FUNCTION_BLOCK Q_ChildPosition (* Command change child position ( Part 6 - F.16 ) *)
  (* Standard: ISO 11783-6; Description: The Change Child Location command is used to change the absolute position of an object. Return values iso_s16 - E_NO_ERR - OK - E_OVERFLOW - buffer overflow - E_NOACT - Command not possible in current state - E_NO_INSTANCE - No VT client available *)
  (* Version 1.0, 2022-07-08, franz *)
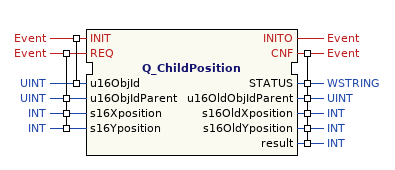
  EVENT_INPUT
    INIT WITH u16ObjId; (* Service Initialization *)
    REQ WITH u16ObjIdParent, s16Xposition, s16Yposition; (* Service Request *)
  END_EVENT
  EVENT_OUTPUT
    INITO; (* Initialization Confirm *)
    CNF WITH STATUS, s16OldYposition, u16OldObjIdParent, s16OldXposition, result; (* Confirmation of Requested Service *)
  END_EVENT
  VAR_INPUT
    u16ObjId : UINT; (* Object ID *)
    u16ObjIdParent : UINT; (* Parent object ID *)
    s16Xposition : INT; (* New X position relative to the top left corner of parent object *)
    s16Yposition : INT; (* New Y position relative to the top left corner of parent object *)
  END_VAR
  VAR_OUTPUT
    STATUS : WSTRING; (* Service Status *)
    u16OldObjIdParent : UINT; (* Old Parent object ID *)
    s16OldXposition : INT; (* Old X position relative to the top left corner of parent object *)
    s16OldYposition : INT; (* Old Y position relative to the top left corner of parent object *)
    result : INT; (* retval see description *)
  END_VAR
END_FUNCTION_BLOCK
